FUNCTION_BLOCK FB_Slitter EXTENDS FB_BASE IMPLEMENTS I_UnitState
VAR_INPUT
	Batch		: ULINT;
	Inspect		: BOOL;					// run routine without cut; just inspect
	InspectCmd	: ST_InspectCommands;
	TubeHmi		: ST_TubeParameters;	// used for manual commands
END_VAR
VAR_IN_OUT
	Tube		: ST_TubeParameters;
END_VAR
VAR_OUTPUT 
	FilesLoaded		: BOOL;
	BatchOut		: ULINT;
	CounterOut		: ULINT;
	CountFailedOut	: UINT;
	Status			: INT; 	// 0 = idle, 1 = processing, 2 = pass, 3 = fail, 4 = no detect
END_VAR
VAR
	Mandrel				: FB_Mandrel;
	MandrelParameters	: ST_MandrelParameters;
	Camera				: FB_Camera;
	CameraParameters	: ST_CameraParameters;
	Cutter				: FB_Cutter;
	CutterParameters 	: ST_CutterParameters;
	Ejector				: FB_Ejector;
	EjectorParameters	: ST_EjectorParameters;
	EjectState			: INT;
	Eject				: BOOL;
	
	Manual		: ST_ManualCommands;
	bBusy		: BOOL;	
	bCalibration: BOOL;
	strJobName	: STRING;	// for manual override of which camera program is used
	nIndex		: INT;
	PreviousTubeIndex	: INT;
	fbFileOpen	: FB_FileOpen;
	fbFileWrite	: FB_FileWrite;
	fbFileClose	: FB_FileClose;
	fbLocalSystemTime	: FB_LocalSystemTime;
	bDecrementSpindle: BOOL;
	bIncrementSpindle: BOOL;
	bInspect: BOOL;
	bInspectComplete: BOOL;
	nCalibrationCounter : INT;
	CalibrationArrayX	: ARRAY[0..CalMax] OF LREAL;
	CalibrationArrayY	: ARRAY[0..CalMax] OF LREAL;
	AverageX 			: LREAL;
	AverageY 			: LREAL;
	
	fbXmlSrvRead		: FB_XmlSrvRead;
	fbXmlSrvWrite		: FB_XmlSrvWrite;

	fbMessageSaved		: FB_TcMessage;
		
END_VAR
VAR CONSTANT
	CalMax	: INT := 9;
END_VAR
VAR PERSISTENT
	Counter		: UINT;
	CountFailed	: UINT;
END_VAR


SUPER^();

IF eState <> E_PMLState.ePMLState_Undefined THEN
	Mandrel.MonitorParameters();
	Camera.MonitorParameters();
	Cutter.MonitorParameters();
	Ejector.MonitorParameters();
END_IF

Mandrel.ConvertVaccum();
Mandrel.TubeParameters := Tube;

IF Batch <> BatchOut THEN
	BatchOut := Batch;
	Counter := 0;
	CountFailed := 0;
END_IF

CounterOut := Counter;
CountFailedOut := CountFailed;

Camera.TubeParameters := Tube;

CASE eState OF
	E_PMLState.ePMLState_Idle: Status := 0;
	E_PMLState.ePMLState_Starting: Status := 1;
	(* put in executing to get fast answer - don't wait for execute to finish
	E_PMLState.ePMLState_Completing:
		IF Camera.Pass THEN
			Status := 2;
		ELSIF Camera.Fail THEN
			Status := 3;
		ELSIF ...
			Status := 4;
		END_IF
	*)
END_CASE

METHOD FB_init : BOOL
VAR_INPUT
	bInitRetains : BOOL; // if TRUE, the retain variables are initialized (warm start / cold start)
	bInCopyCode : BOOL;  // if TRUE, the instance afterwards gets moved into the copy code (online change)
END_VAR
IF NOT fbMessageSaved.EqualsToEventEntryEx(stOther := TC_EVENTS.SlitterEvents.ParametersSaved) THEN
	fbMessageSaved.CreateEx(TC_EVENTS.SlitterEvents.ParametersSaved, 0);
END_IF
END_METHOD

METHOD M_Aborting
M_StateComplete();

bBusy := FALSE;
bCalibration := FALSE;
Cutter.Abort();
Ejector.Abort();
Mandrel.Abort();
M_CalibrateCamera(Execute := FALSE);
Eject := FALSE;
EjectState := 0;
nCalibrationCounter := 0;

Manual.bCameraCalibrate := FALSE;
Manual.bCameraComputePeak := FALSE;
Manual.bCameraInspect := FALSE;
Manual.bCameraRawData := FALSE;
Manual.bCameraTrigger := FALSE;
Manual.bCutSample := FALSE;
Manual.bCutterDisable := FALSE;
Manual.bCutterHome := FALSE;
Manual.bCutterMoveAbs := FALSE;
Manual.bCutterReset := FALSE;
Manual.bEjectAxisEnableToggle := FALSE;
Manual.bEjectAxisFailPosition := FALSE;
Manual.bEjectAxisHomePosition := FALSE;
Manual.bEjectAxisPassPosition := FALSE;
Manual.bEjectAxisReset := FALSE;
Manual.bEjectBlowOff := FALSE;
Manual.bEjectReset := FALSE;
Manual.bEjectSamplePass := FALSE;
Manual.bEjectSampleFail := FALSE;
Manual.bEjectVacuum := FALSE;
Manual.bEjectZExtend := FALSE;
Manual.bEjectZNeutral := FALSE;
Manual.bEjectZOff := FALSE;
Manual.bEjectZRetract := FALSE;
Manual.bLowerMandrel := FALSE;
Manual.bMandrelReset := FALSE;
Manual.bMandrelSpindleRotate := FALSE;
Manual.bMandrelSpindleToggle := FALSE;
Manual.bMandrelXEnableToggle := FALSE;
Manual.bMandrelYEnableToggle := FALSE;
Manual.bMoveToCutPosition := FALSE;
Manual.bMoveToEjectPosition := FALSE;
Manual.bMoveToInspectPosition := FALSE;
Manual.bMoveToLoadPosition := FALSE;
Manual.bRaiseMandrel := FALSE;
Manual.bSaveMandrelParameters := FALSE;
Manual.bToggleMandrelVacuum := FALSE;
Manual.bVacuumAxisToggleEnable := FALSE;
Manual.bVacuumAxisMove := FALSE;
Manual.bVacuumAxisReset := FALSE;
END_METHOD

METHOD M_CalibrateCamera : INT;
VAR_INPUT
	Execute			: BOOL;
END_VAR
VAR_INST
	rTrig			: R_TRIG;
	nIndex			: INT;
	Position		: LREAL;
	debug			: INT;
	debug1			: INT;
	debug2			: INT;
END_VAR
rTrig(CLK := Execute);
IF rTrig.Q THEN
	nIndex := 10;
	Mandrel.MoveToInspectPosition(Execute := FALSE, InspectPositionX := Tube.InspectPositionX, InspectPositionY := Tube.InspectPositionY);
	Mandrel.MoveToLoadPosition(Execute := FALSE);
	Mandrel.MoveXAbs(Execute := FALSE, Position := 0);
	Mandrel.MoveYAbs(Execute := FALSE, Position := 0);
	Camera.TriggerCamera(Execute := FALSE);
	bCalibration := TRUE;
END_IF

IF NOT Execute THEN
	debug := debug + 1;
	nIndex := 0;
END_IF

CASE nIndex OF
	0: // idle state
		M_CalibrateCamera := 0;
		bCalibration := FALSE;
	10: // move to first inspection position
		IF Mandrel.MoveToInspectPosition(Execute := TRUE, InspectPositionX := Tube.InspectPositionX, InspectPositionY := Tube.InspectPositionY) = 1 THEN
			Mandrel.MoveToInspectPosition(Execute := FALSE, InspectPositionX := Tube.InspectPositionX, InspectPositionY := Tube.InspectPositionY);
			nIndex := 20;
		ELSIF Mandrel.MoveToInspectPosition(Execute := TRUE, InspectPositionX := Tube.InspectPositionX, InspectPositionY := Tube.InspectPositionY) = -1 THEN
			Mandrel.MoveToInspectPosition(Execute := FALSE, InspectPositionX := Tube.InspectPositionX, InspectPositionY := Tube.InspectPositionY);
			nIndex := 100;
		END_IF
	20: // trigger the camera
		IF Camera.TriggerCamera(Execute := TRUE) THEN
			Camera.PatternX1 := Camera.PatternMatchX;
			Camera.PatternY1 := Camera.PatternMatchY;
			Camera.TriggerCamera(Execute := FALSE);
			nIndex := 30;
		END_IF
	30: // move to second position in x
		Position := Tube.InspectPositionX + Camera.CalibrationDistance; 
		IF Mandrel.MoveXAbs(Execute := TRUE, Position := Position) = 1 THEN
			Mandrel.MoveXAbs(Execute := FALSE, Position := Position);
			nIndex := 40;
		ELSIF Mandrel.MoveXAbs(Execute := TRUE, Position := Position) = -1 THEN
			Mandrel.MoveXAbs(Execute := FALSE, Position := Position);
			nIndex := 100;
		END_IF
	40: // trigger the camera
		IF Camera.TriggerCamera(Execute := TRUE) THEN
			Camera.PatternX2 := Camera.PatternMatchX;
			Camera.PatternY2 := Camera.PatternMatchY;
			Camera.TriggerCamera(Execute := FALSE);
			nIndex := 50;
		END_IF
	45: // 
		Mandrel.MoveYAbs(Execute := FALSE, Position := 0);
		nIndex := 50;
	50: // move to the third position in y
		Position := Tube.InspectPositionY + Camera.CalibrationDistance; 
		IF Mandrel.MoveYAbs(Execute := TRUE, Position := Position) = 1 THEN
			Mandrel.MoveYAbs(Execute := FALSE, Position := Position);
			nIndex := 60;
		ELSIF Mandrel.MoveYAbs(Execute := TRUE, Position := Position) = -1 THEN
			Mandrel.MoveYAbs(Execute := FALSE, Position := Position);
			nIndex := 100;
		END_IF
	60: // trigger camera
		IF Camera.TriggerCamera(Execute := TRUE) THEN
			Camera.PatternX3 := Camera.PatternMatchX;
			Camera.PatternY3 := Camera.PatternMatchY;
			Camera.TriggerCamera(Execute := FALSE);
			nIndex := 70;
		END_IF
	70: // Calculate the pitch
		Camera.Calibrate();
		nIndex := 80; 
	80: // return to load position	
		IF Mandrel.MoveToLoadPosition(Execute := TRUE) <> 0 THEN
			Mandrel.MoveToLoadPosition(Execute := FALSE);
			nIndex := 90;
		END_IF
	90: // done state
		M_CalibrateCamera := 1;
	 
	100: // error state
		M_CalibrateCamera := -1;
	
END_CASE
END_METHOD

METHOD M_Clearing
CASE eMode OF
	E_PMLProtectedUnitMode.ePMLProtUnitMode_Manual: M_ClearingManual();
	
	E_PMLProtectedUnitMode.ePMLProtUnitMode_Production: M_ClearingProduction();
END_CASE
END_METHOD

METHOD M_ClearingManual : BOOL
VAR_INPUT
END_VAR
M_StateComplete();
//M_ClearingManual := TRUE;
END_METHOD

METHOD M_ClearingProduction : BOOL
VAR_INPUT
END_VAR
CASE nState OF
	0:	// reset the variables
		Mandrel.Clear(Execute := FALSE);
		Cutter.Clear(Execute := FALSE);
		Ejector.Reset(Execute := FALSE);
		nState := 10;
	10: // reset the cutter
		IF Cutter.Clear(Execute := TRUE) = 1 THEN
			Cutter.Clear(Execute := FALSE);
			nState := 20;
		END_IF	
	20: // reset the ejector
		IF Ejector.Reset(Execute := TRUE) = 1 THEN
			Ejector.Reset(Execute := FALSE);
			nState := 30;		END_IF

	30: // reset the different objects
		IF Mandrel.Clear(Execute := TRUE) = 1 THEN
			Mandrel.Clear(Execute := FALSE);
			nState := 40;
		END_IF
	40:	// done state
		M_StateComplete();
END_CASE
END_METHOD


METHOD M_Complete
END_METHOD

METHOD M_Completing

VAR
	EjectSample: INT;
END_VAR
IF eMode = E_PMLProtectedUnitMode.ePMLProtUnitMode_Production THEN
	CASE EjectState OF
		0: // wait for eject command
			M_StateComplete();
		10: // execute the eject pass sequence
			EjectSample := Ejector.EjectSamplePass(Execute := TRUE);
			IF EjectSample = 1 THEN
				Eject := FALSE;
				Ejector.EjectSamplePass(Execute := FALSE);
				EjectState := 0;
			ELSIF EjectSample = -1 THEN
				Eject := FALSE;
				EjectState := 0;
				Ejector.EjectSamplePass(Execute := FALSE);
			END_IF
		20: // execute the eject fail sequence
			EjectSample := Ejector.EjectSampleFail(Execute := TRUE);
			IF EjectSample = 1 THEN
				Eject := FALSE;
				Ejector.EjectSampleFail(Execute := FALSE);
				EjectState := 0;
			ELSIF EjectSample = -1 THEN
				Eject := FALSE;
				EjectState := 0;
				Ejector.EjectSampleFail(Execute := FALSE);
			END_IF
	END_CASE
ELSE
	M_StateComplete();
END_IF
END_METHOD

METHOD M_Execute
VAR_INST
	Result					: INT;
END_VAR
VAR
	CutPositionY 			: LREAL;
	VelocityY 				: LREAL;
	MoveToCutPosition 		: INT;
	MoveToInspectPosition 	: INT;
	MoveToEjectPosition 	: INT;
	MoveToLoadPosition 		: INT;
	CutSample				: INT;
	EjectSample 			: INT;

	CameraIndex 			: INT;
	FileName				: STRING;
	FilePath				: STRING;
	RotateDistance			: LREAL;
END_VAR
VAR_INST
	StrResult				: STRING(255);
	SampleLowered			: BOOL;
	LiftTon					: TON := (PT := T#500MS);
	VacuumSensorTON			: TON := (PT := T#2S);
	hFile					: UINT;
	AttemptCounter			: INT;
	Pass					: BOOL;
	Message					: STRING(255);
END_VAR
Eject := FALSE;
fbLocalSystemTime(
	sNetId := '',
	bEnable := TRUE,
	dwCycle := 1);

IF eMode = E_PMLProtectedUnitMode.ePMLProtUnitMode_Production THEN
	CASE nState OF
		0: // do we need to write to the camera?
			AttemptCounter := 0;
			bDecrementSpindle:= FALSE;
			bIncrementSpindle:= FALSE;
			bInspect:= FALSE;
			bInspectComplete:= FALSE;

			SampleLowered := FALSE;
			VacuumSensorTON(IN := FALSE);
			Result := Camera.SelectCameraProgram(Execute := TRUE);
			IF Result = 1 THEN
				Camera.SelectCameraProgram(Execute := FALSE);
				nState := 5;
			ELSIF Result = -1 THEN
				Camera.SelectCameraProgram(Execute := FALSE);
				Message := 'Camera failed to read/write to modbus.';
				nState := 666;
			END_IF
		5: // move the vacuum axis to the correct location
			IF Mandrel.MoveToVacPosition(Execute := TRUE) THEN
				Mandrel.MoveToVacPosition(Execute := FALSE);
				nState := 10;
			END_IF
		10: // turn on mandrel vacuum and move to cut position
			Mandrel.MandrelVacuum := TRUE;
			IF Mandrel.LowerSample() = 1 THEN
				SampleLowered := TRUE;
				nState := 11;
			END_IF
		11: // wait for vacuum sensor to detect the tube
			VacuumSensorTON(IN := TRUE);
			IF Mandrel.VacuumSensor > Tube.VacuumThreshold THEN
				nState := 15;
				VacuumSensorTON(IN := FALSE);
			END_IF
			IF VacuumSensorTON.Q THEN
				Mandrel.MandrelVacuum := FALSE;
				nState := 110;
				VacuumSensorTON(IN := FALSE);
			END_IF
		15: // move to cut position
			MoveToCutPosition := Mandrel.MoveToCutPosition(Execute := TRUE, CutPositionX := Tube.CutPositionX, CutPositionY := Tube.CutPositionY);
			IF MoveToCutPosition = 1 AND SampleLowered THEN
				Mandrel.MoveToCutPosition(Execute := FALSE, CutPositionX := Tube.CutPositionX, CutPositionY := Tube.CutPositionY);
				nState := 20;
				SampleLowered := FALSE;
			ELSIF MoveToCutPosition = -1 THEN
				Mandrel.MoveToCutPosition(Execute := FALSE, CutPositionX := Tube.CutPositionX, CutPositionY := Tube.CutPositionY);
				nState := 666;
				Message := 'Mandrel failed to move.';
				SampleLowered := FALSE;
			END_IF
		20: // make a cut unless we are just inspecting
			IF Inspect THEN
				nState := 30;
			ELSE
				CutSample := Cutter.CutSample(Execute := TRUE);
				IF CutSample = 1 THEN
					Cutter.CutSample(Execute := FALSE);
					nState := 30;
				ELSIF CutSample = -1 THEN
					Cutter.CutSample(Execute := FALSE);
					nState := 666;
				END_IF
			END_IF
		30: // raise sample
			// move to inspect position
			Mandrel.LiftSample();
			MoveToInspectPosition := Mandrel.MoveToInspectPosition(Execute := TRUE, InspectPositionX := Tube.InspectPositionX, InspectPositionY := Tube.InspectPositionY);
			IF MoveToInspectPosition = 1 THEN
				Mandrel.MoveToInspectPosition(Execute := FALSE, InspectPositionX := Tube.InspectPositionX, InspectPositionY := Tube.InspectPositionY);
				nState := 35;
			ELSIF MoveToInspectPosition = -1 THEN
				Mandrel.MoveToInspectPosition(Execute := FALSE, InspectPositionX := Tube.InspectPositionX, InspectPositionY := Tube.InspectPositionY);
				nState := 666;
			END_IF
		35: // add 500 ms delay for lifter
			LiftTON.IN := TRUE;
			IF LiftTON.Q THEN
				LiftTON.IN := FALSE;
				IF Inspect THEN
					nState := 36;
				ELSE
					nState := 40;
				END_IF
			END_IF
			LiftTON();
		36: // Inspect under manual control
			Result := Camera.Inspect(Execute := TRUE);
			IF Result = 1 THEN
				nState := 37;
				Camera.Inspect(Execute := FALSE);
				IF Camera.Pass THEN
					Status := 2;
				ELSE
					Status := 3;
				END_IF
			ELSIF Result = -1 THEN
				Status := 4;
				nState := 37;
			END_IF
			//nState := 37;
		37: // wait for command
			IF bDecrementSpindle THEN
				bDecrementSpindle := FALSE;
				nState := 39;
			ELSIF bIncrementSpindle THEN
				bIncrementSpindle := FALSE;
				nState := 38;
			ELSIF bInspect THEN
				bInspect := FALSE;
				nState := 36;
			ELSIF bInspectComplete THEN
				bInspectComplete := FALSE;
				nState := 70;
			END_IF
		38: // increment spindle
			IF Mandrel.RotateSpindle(Execute := TRUE, Distance := Mandrel.SpindleIncrement ) <> 0 THEN
				Mandrel.RotateSpindle(Execute := FALSE, Distance := Mandrel.SpindleIncrement);
				nState := 37;
			END_IF
		39: // decrement spindle
			IF Mandrel.RotateSpindle(Execute := TRUE, Distance := -1 * Mandrel.SpindleIncrement) <> 0 THEN
				Mandrel.RotateSpindle(Execute := FALSE, Distance := -1 * Mandrel.SpindleIncrement);
				nState := 37;
			END_IF
			
		40: // inspect
			Result := Camera.Inspect(Execute := TRUE);
			IF Result = 1 THEN
				Camera.Inspect(Execute := FALSE);
				IF Camera.Pass THEN
					Mandrel.MandrelVacuum := FALSE;
					IF Manual.bCalibrateMandrel THEN
						CalibrationArrayX[nCalibrationCounter] := Camera.DeltaXmmWithOffset;
						CalibrationArrayY[nCalibrationCounter] := Camera.DeltaYmmWithOffset;
						nCalibrationCounter := nCalibrationCounter + 1;
						IF nCalibrationCounter > CalMax THEN
							MandrelCalibration();
							Manual.bCalibrateMandrel := FALSE;
							nCalibrationCounter := 0;
						END_IF
					END_IF
					Pass := TRUE;
					nState := 50;	// passed -> go to eject pass station
					Status := 2;
				ELSE
					Mandrel.MandrelVacuum := FALSE;
					Pass := FALSE;
					nState := 50;	// failed -> go to eject fail station
					Status := 3;
				END_IF
			ELSIF Result = -1 THEN	// couldn't find the pattern; need to advance the counter and retry
				AttemptCounter := AttemptCounter + 1;
				Camera.Inspect(Execute := FALSE);
				IF AttemptCounter > 3 THEN	// error
					nState := 70;			// error out
					Status := 4;
				ELSE						// advance the motor a bit and retry
					nState := 45;
				END_IF
			END_IF
		45: // advance the tube a bit and then go and retry the process
			Result := Mandrel.MoveXRel(Execute := TRUE, Distance := 1);
			IF Result = 1 THEN
				Mandrel.MoveXRel(Execute := FALSE, Distance := 1);
				nState := 35;
			END_IF
			
		50: // move to eject position		
			MoveToEjectPosition := Mandrel.MoveToEjectPosition(Execute := TRUE, EjectPositionX := Tube.EjectPositionX, EjectPositionY := Tube.EjectPositionY);
			IF MoveToEjectPosition = 1 THEN
				Mandrel.MoveToEjectPosition(Execute := FALSE, EjectPositionX := Tube.EjectPositionX, EjectPositionY := Tube.EjectPositionY);
				nState := 60;
			ELSIF MoveToEjectPosition = -1 THEN
				Mandrel.MoveToEjectPosition(Execute := FALSE, EjectPositionX := Tube.EjectPositionX, EjectPositionY := Tube.EjectPositionY);
				nState := 666;
			END_IF
		60: // do the eject sequence 
			Eject := TRUE;		
			// wait for the system to retract
			IF Ejector.IsEjectZExtend THEN
				nState := 65;
			END_IF
		65: // wait for ejector actuator to be clear to retract the mandrel
			IF Ejector.IsEjectZRetract THEN
				nState := 70;
			END_IF 
		70: // move to load position
			Mandrel.MandrelVacuum := FALSE;

			IF Mandrel.LowerSample() = 1 THEN
				SampleLowered := TRUE;
			END_IF
			IF Manual.bCalibrateMandrel THEN
				IF Mandrel.SpindleOffset >= 0 THEN
					RotateDistance := (360.0 / (INT_TO_LREAL(CalMax)+1.0)) - Mandrel.SpindleOffset;
				ELSE
					RotateDistance := -1 * ( (360.0 / (INT_TO_LREAL(CalMax)+1.0)) + Mandrel.SpindleOffset);
				END_IF
				IF Mandrel.RotateSpindle(Execute := TRUE, Distance := RotateDistance) <> 0 THEN
					Mandrel.RotateSpindle(Execute := FALSE, Distance := RotateDistance);
					nState := 75;
				END_IF
			ELSE
				nState := 75;			
			END_IF
		75: // move to load position cont'd
			IF Mandrel.LowerSample() = 1 THEN
				SampleLowered := TRUE;
			END_IF

			MoveToLoadPosition := Mandrel.MoveToLoadPosition(Execute := TRUE);
			IF MoveToLoadPosition = 1 AND SampleLowered THEN
				Mandrel.MoveToLoadPosition(Execute := FALSE);
				SampleLowered := FALSE;
				nState := 80;
			ELSIF MoveToLoadPosition = -1 THEN
				SampleLowered := FALSE;
				Mandrel.MoveToLoadPosition(Execute := FALSE);
				nState := 666;
			END_IF
		80: // check if vacuum is off
			IF Mandrel.VacuumSensor < Tube.VacuumThreshold THEN
				nState := 90;
				Mandrel.MandrelVacuum := FALSE;
			END_IF
		90:	// increment counters state
			IF NOT Inspect THEN			
				Counter := Counter + 1;
				IF NOT Camera.Pass THEN
					CountFailed := CountFailed + 1;
				END_IF
				nState := 100;
			ELSE
				nState := 110;
			END_IF			
		100: // save to file
			FileName := CONCAT(ULINT_TO_STRING(Batch), '.txt');
			FilePath := CONCAT('D:\',FileName);
			fbFileOpen(
				sNetId := '',
				sPathName := FilePath,
				nMode := FOPEN_MODEAPPEND,
				ePath := E_OpenPath.PATH_GENERIC,
				hFile => hFile,
				bExecute := TRUE);
			IF NOT fbFileOpen.bBusy THEN
				fbFileOpen(
					sNetId := '',
					sPathName := FilePath,
					nMode := FOPEN_MODEAPPEND,
					ePath := E_OpenPath.PATH_GENERIC,
					bExecute := FALSE);
				nState := 101;
			END_IF
			IF fbFileOpen.bError THEN
				fbFileOpen(
					sNetId := '',
					sPathName := FilePath,
					nMode := FOPEN_MODEAPPEND,
					ePath := E_OpenPath.PATH_GENERIC,
					bExecute := FALSE);
				nState := 102;				
			END_IF
		101: // write data to file	
			StrResult := '';		
			StrResult := CONCAT(ULINT_TO_STRING(Batch), ', ');
			StrResult := CONCAT(StrResult, UINT_TO_STRING(Counter));
			StrResult := CONCAT(StrResult, ', ');
			// add the system time
			IF fbLocalSystemTime.bValid THEN
				StrResult := CONCAT(StrResult, SYSTEMTIME_TO_STRING(fbLocalSystemTime.systemTime));
				StrResult := CONCAT(StrResult, ', ');
			END_IF
			IF Camera.Pass THEN
				StrResult := CONCAT(StrResult, 'PASS, ');
			ELSIF Camera.Fail THEN
				StrResult := CONCAT(StrResult, 'FAIL, ');
			ELSIF Camera.NoDetect THEN
				StrResult := CONCAT(StrResult, 'NO DETECT, ');
			END_IF
			IF NOT Camera.NoDetect THEN
				StrResult := CONCAT(StrResult, 'x := ');
				StrResult := CONCAT(StrResult, REAL_TO_STRING(Camera.DeltaXmmWithOffset));
				StrResult := CONCAT(StrResult, ', y := ');
				StrResult := CONCAT(StrResult, REAL_TO_STRING(Camera.DeltaYmmWithOffset));
				StrResult := CONCAT(StrResult, ', length := ');
				StrResult := CONCAT(StrResult, REAL_TO_STRING(Camera.CutLengthWithOffset));
			ELSE
				StrResult := CONCAT(StrResult, 'x := not detected');
				StrResult := CONCAT(StrResult, ', y := not detected');
				StrResult := CONCAT(StrResult, ', length := not detected');			
			END_IF
			StrResult := CONCAT(StrResult, '$r$n');
			fbFileWrite(
				sNetId := '',
				hFile := hFile,
				pWriteBuff := ADR(StrResult),
				cbWriteLen := INT_TO_UINT(LEN(StrResult)),
				bExecute := TRUE
			);
			IF NOT fbFileWrite.bBusy THEN
				nState := 102;
				fbFileWrite(bExecute := FALSE);
			END_IF
			IF fbFileWrite.bError THEN
				nState := 102;
				fbFileWrite(bExecute := FALSE);
			END_IF
		102: // file close
			fbFileClose(
				sNetId := '',
				hFile := hFile,
				bExecute := TRUE);
			IF NOT fbFileClose.bBusy THEN
				fbFileClose(bExecute := FALSE);
				nState := 110;
			END_IF
			IF fbFileClose.bError THEN
				fbFileClose(bExecute := FALSE);
				nState := 110;
			END_IF
		110: // done state
			M_StateComplete();
	END_CASE
	
	CASE EjectState OF
		0: // wait for eject command
			Ejector.EjectSamplePass(Execute := FALSE);
			Ejector.EjectSampleFail(Execute := FALSE);
			IF Eject AND Pass THEN
				EjectState := 10;
			ELSIF Eject AND NOT Pass THEN
				EjectState := 20;
			END_IF
		10: // execute the eject pass sequence
			EjectSample := Ejector.EjectSamplePass(Execute := TRUE);
			IF EjectSample = 1 THEN
				Eject := FALSE;
				Ejector.EjectSamplePass(Execute := FALSE);
				EjectState := 0;
			ELSIF EjectSample = -1 THEN
				Eject := FALSE;
				EjectState := 0;
				Ejector.EjectSamplePass(Execute := FALSE);
			END_IF
		20: // execute the eject fail sequence
			EjectSample := Ejector.EjectSampleFail(Execute := TRUE);
			IF EjectSample = 1 THEN
				Eject := FALSE;
				Ejector.EjectSampleFail(Execute := FALSE);
				EjectState := 0;
			ELSIF EjectSample = -1 THEN
				Eject := FALSE;
				EjectState := 0;
				Ejector.EjectSampleFail(Execute := FALSE);
			END_IF

	END_CASE
ELSIF eMode = E_PMLProtectedUnitMode.ePMLProtUnitMode_Manual THEN
	M_Manual();
END_IF
END_METHOD


METHOD M_Held
END_METHOD


METHOD M_Holding
END_METHOD


METHOD M_Idle
END_METHOD

METHOD M_Manual : BOOL
VAR_INPUT
END_VAR
VAR_INST
	Operational	: BOOL;
	Result		: INT;
	TON			: TON := (PT := T#5S);
	x			: INT;
END_VAR

IF Manual.bCameraCalibrate THEN
	bBusy := TRUE;
	IF M_CalibrateCamera(Execute := TRUE) <> 0 THEN
		M_CalibrateCamera(Execute := FALSE);
		bBusy := FALSE;
		Manual.bCameraCalibrate := FALSE;
	END_IF
END_IF

IF Manual.bCameraComputePeak THEN
	bBusy := TRUE;
	IF Camera.Compute(Execute := TRUE) = 1 THEN
		bBusy := FALSE;
		Camera.Compute(Execute := FALSE);
		Manual.bCameraComputePeak := FALSE;
	END_IF
END_IF

IF Manual.bCameraInspect THEN
	bBusy := TRUE;
	IF Camera.Inspect(Execute := TRUE) = 1 THEN
		Camera.Inspect(Execute := FALSE);
		Manual.bCameraInspect := FALSE;
		bBusy := FALSE;
	END_IF
END_IF	

IF Manual.bCameraRawData THEN
	bBusy := TRUE;
	IF Camera.GetCameraData() <> 0 THEN
		bBusy := FALSE;
		Manual.bCameraRawData := FALSE;
	END_IF
END_IF

IF Manual.bCameraSelectTube THEN
	bBusy := TRUE;
	Result := Camera.SelectCameraProgram(Execute := TRUE);
	IF Result = 1 THEN
		bBusy := FALSE;
		Manual.bCameraSelectTube := FALSE;
		Camera.SelectCameraProgram(Execute := FALSE);
	ELSIF Result = -1 THEN
		bBusy := FALSE;
		Manual.bCameraSelectTube := FALSE;
		Camera.SelectCameraProgram(Execute := FALSE);
		x := x + 1;
	END_IF
END_IF

IF Manual.bCameraTrigger THEN
	bBusy := TRUE;
	IF Camera.TriggerCamera(Execute := TRUE) THEN
		Camera.TriggerCamera(Execute := FALSE);
		bBusy := FALSE;
		Manual.bCameraTrigger := FALSE;
	END_IF
END_IF

IF Manual.bCutSample THEN
	bBusy := TRUE;
	IF Cutter.CutSample(Execute := TRUE) <> 0 THEN
		Cutter.CutSample(Execute := FALSE);
		Manual.bCutSample := FALSE;
		bBusy := FALSE;
	END_IF
END_IF

IF Manual.bCutterDisable THEN
	IF NOT bBusy THEN
		Operational := Cutter.IsEnabled;
		TON(IN := TRUE);
	END_IF
	bBusy := TRUE;
	IF Operational THEN
		IF Cutter.Disable() THEN
			TON(IN := FALSE);
			bBusy := FALSE;
			Manual.bCutterDisable := FALSE;
		END_IF
	ELSE
		IF Cutter.Enable() OR TON.q	THEN
			bBusy := FALSE;
			TON(IN := FALSE);
			Manual.bCutterDisable := FALSE;
		END_IF
	END_IF
	TON();
END_IF

IF Manual.bCutterHome THEN
	bBusy := TRUE;
	IF Cutter.Home(Execute := TRUE) <> 0 THEN
		bBusy := FALSE;
		Cutter.Home(Execute := FALSE);
		Manual.bCutterHome := FALSE;
	END_IF
END_IF

IF Manual.bCutterMoveAbs THEN
	bBusy := FALSE;
	IF Cutter.MoveAbs(Execute := TRUE) <> 0 THEN
		bBusy := FALSE;
		Cutter.MoveAbs(Execute := FALSE);
		Manual.bCutterMoveAbs := FALSE;
	END_IF
END_IF

IF Manual.bCutterReset THEN
	bBusy := TRUE;
	IF Cutter.Reset(Execute := TRUE) <> 0 THEN
		bBusy := FALSE;
		Manual.bCutterReset := FALSE;
		Cutter.Reset(Execute := FALSE);
	END_IF
END_IF

IF Manual.bEjectBlowOff THEN
	Ejector.BlowOff := NOT Ejector.BlowOff;
	Manual.bEjectBlowOff := FALSE;
END_IF

IF Manual.bEjectSamplePass THEN
	bBusy := TRUE;
	IF Ejector.EjectSamplePass(Execute := TRUE) = 1 THEN
		Ejector.EjectSamplePass(Execute := FALSE);
		Manual.bEjectSamplePass := FALSE;
		bBusy := FALSE;
	END_IF
END_IF

IF Manual.bEjectSampleFail THEN
	bBusy := TRUE;
	IF Ejector.EjectSampleFail(Execute := TRUE) = 1 THEN
		Ejector.EjectSampleFail(Execute := FALSE);
		Manual.bEjectSampleFail := FALSE;
		bBusy := FALSE;
	END_IF
END_IF

IF Manual.bEjectVacuum THEN
	Ejector.PickUpVacuum := NOT Ejector.PickUpVacuum;
	Manual.bEjectVacuum := FALSE;
END_IF
(*
	bEjectAxisPassPosition	: BOOL;
	bEjectAxisHomePosition	: BOOL;
	bEjectAxisFailPosition	: BOOL;
	bEjectAxisEnable		: BOOL;
	bEjectAxisDisabe		: BOOL;
	bEjectAxisReset			: BOOL;
	bEjectSamplePass		: BOOL;
	bEjectSampleFail		: BOOL;
*)
IF Manual.bEjectAxisEnableToggle THEN
	IF NOT bBusy THEN
		Operational := Ejector.axis.IsEnabled;
	END_IF
	bBusy := TRUE;
	IF Operational THEN
		IF Ejector.axis.Disable() THEN
			bBusy := FALSE;
			Manual.bEjectAxisEnableToggle := FALSE;
		END_IF
	ELSE
		IF Ejector.axis.Enable() THEN
			bBusy := FALSE;
			Manual.bEjectAxisEnableToggle := FALSE;
		END_IF		
	END_IF
END_IF

IF Manual.bEjectAxisFailPosition THEN
	bBusy := TRUE;
	IF Ejector.axis.AbsMove(Execute := TRUE, 
		Position := Ejector.EjectAxisFailPosition, 
		Velocity := Ejector.EjectAxisVelocity) THEN
			Ejector.axis.AbsMove(Execute := FALSE, Position := Ejector.EjectAxisFailPosition, Velocity := Ejector.EjectAxisVelocity);	
			bBusy := FALSE;
			Manual.bEjectAxisFailPosition := FALSE;
	END_IF
END_IF

IF Manual.bEjectAxisHomePosition THEN
	bBusy := TRUE;
	IF Ejector.axis.AbsMove(Execute := TRUE, 
		Position := Ejector.EjectAxisHomePosition, 
		Velocity := Ejector.EjectAxisVelocity) THEN
			Ejector.axis.AbsMove(Execute := FALSE, Position := Ejector.EjectAxisHomePosition, Velocity := Ejector.EjectAxisVelocity);
			bBusy := FALSE;
			Manual.bEjectAxisHomePosition := FALSE;
	END_IF
END_IF

IF Manual.bEjectAxisPassPosition THEN
	bBusy := TRUE;
	IF Ejector.axis.AbsMove(Execute := TRUE, 
		Position := Ejector.EjectAxisPassPosition, 
		Velocity := Ejector.EjectAxisVelocity) THEN
			Ejector.axis.AbsMove(Execute := FALSE, Position := Ejector.EjectAxisPassPosition, Velocity := Ejector.EjectAxisVelocity);
			bBusy := FALSE;
			Manual.bEjectAxisPassPosition := FALSE;
	END_IF
END_IF

IF Manual.bEjectAxisReset THEN
	bBusy := TRUE;
	IF Ejector.axis.Reset(Execute := TRUE) THEN
		Ejector.axis.Reset(Execute := FALSE);
		bBusy := FALSE;
		Manual.bEjectAxisReset := FALSE;
	END_IF
END_IF

IF Manual.bEjectReset THEN
	bBusy := TRUE;
	IF Ejector.Reset(TRUE) = 1 THEN
		Ejector.Reset(FALSE);
		bBusy := FALSE;
		Manual.bEjectReset := FALSE;
	END_IF
END_IF

IF Manual.bEjectZExtend THEN
	bBusy := TRUE;
	IF Ejector.zSlide.Extend() = 1 THEN
		bBusy := FALSE;
		Manual.bEjectZExtend := FALSE;
	END_IF
END_IF

IF Manual.bEjectZNeutral THEN
	bBusy := TRUE;
	IF Ejector.zSlide.Neutral() THEN
		bBusy := FALSE;
		Manual.bEjectZNeutral := FALSE;
	END_IF
END_IF

IF Manual.bEjectZRetract THEN
	bBusy := TRUE;
	IF Ejector.zSlide.Retract() = 1 THEN
		bBusy := FALSE;
		Manual.bEjectZRetract := FALSE;
	END_IF
END_IF

IF Manual.bLowerMandrel THEN
	bBusy := TRUE;
	IF Mandrel.LowerSample() = 1 THEN
		bBusy := FALSE;
		Manual.bLowerMandrel := FALSE;
	END_IF
END_IF

IF Manual.bMandrelSpindleRotate THEN
	bBusy := TRUE;
	IF Mandrel.RotateSpindle(Execute := TRUE, Distance := Mandrel.SpindleIncrement) <> 0 THEN
		bBusy := FALSE;
		Mandrel.RotateSpindle(Execute := FALSE, Distance := Mandrel.SpindleIncrement);
		Manual.bMandrelSpindleRotate := FALSE;
	END_IF
END_IF

IF Manual.bMandrelSpindleToggle THEN
	IF NOT bBusy THEN
		Operational := Mandrel.OperationalSpindle;
	END_IF
	bBusy := TRUE;
	IF Operational THEN
		IF Mandrel.DisableSpindle() THEN
			bBusy := FALSE;
			Manual.bMandrelSpindleToggle := FALSE;
		END_IF
	ELSE
		IF Mandrel.EnableSpindle() THEN
			bBusy := FALSE;
			Manual.bMandrelSpindleToggle := FALSE;
		END_IF
	END_IF
END_IF

IF Manual.bMandrelXEnableToggle THEN
	IF NOT bBusy THEN
		Operational := Mandrel.OperationalX;
	END_IF
	bBusy := TRUE;
	IF Operational THEN
		IF Mandrel.DisableX() THEN
			bBusy := FALSE;
			Manual.bMandrelXEnableToggle := FALSE;
		END_IF
	ELSE
		IF Mandrel.EnableX() THEN
			bBusy := FALSE;
			Manual.bMandrelXEnableToggle := FALSE;
		END_IF
	END_IF	
END_IF

IF Manual.bMandrelYEnableToggle THEN
	IF NOT bBusy THEN
		Operational := Mandrel.OperationalY;
	END_IF
	bBusy := TRUE;
	IF Operational THEN
		IF Mandrel.DisableY() THEN
			bBusy := FALSE;
			Manual.bMandrelYEnableToggle := FALSE;
		END_IF
	ELSE
		IF Mandrel.EnableY() THEN
			bBusy := FALSE;
			Manual.bMandrelYEnableToggle := FALSE;
		END_IF
	END_IF		
END_IF

IF Manual.bMandrelReset THEN
	bBusy := TRUE;
	IF Mandrel.Reset(Execute := TRUE) = 1 THEN
		Mandrel.Reset(Execute := FALSE);
		bBusy := FALSE;
		Manual.bMandrelReset := FALSE;
	END_IF
END_IF

IF Manual.bMoveToCutPosition THEN
	bBusy := TRUE;
	IF Mandrel.MoveToCutPosition(Execute := TRUE, CutPositionX := TubeHmi.CutPositionX, CutPositionY := TubeHmi.CutPositionY ) = 1 THEN
		Mandrel.MoveToCutPosition(Execute := FALSE, CutPositionX := TubeHmi.CutPositionX, CutPositionY := TubeHmi.CutPositionY);
		Manual.bMoveToCutPosition := FALSE;
		bBusy := FALSE;
	END_IF
END_IF

IF Manual.bMoveToEjectPosition THEN
	bBusy := TRUE;
	IF Mandrel.MoveToEjectPosition(Execute := TRUE, EjectPositionX := TubeHmi.EjectPositionX, EjectPositionY := TubeHmi.EjectPositionY) = 1 THEN
		Mandrel.MoveToEjectPosition(Execute := FALSE, EjectPositionX := TubeHmi.EjectPositionX, EjectPositionY := TubeHmi.EjectPositionY);
		Manual.bMoveToEjectPosition := FALSE;
		bBusy := FALSE;
	END_IF
END_IF

IF Manual.bMoveToInspectPosition THEN
	bBusy := TRUE;
	IF Mandrel.MoveToInspectPosition(Execute := TRUE, InspectPositionX := TubeHmi.InspectPositionX, InspectPositionY := TubeHmi.InspectPositionY) = 1 THEN
		Mandrel.MoveToInspectPosition(Execute := FALSE, InspectPositionX := TubeHmi.InspectPositionX, InspectPositionY := TubeHmi.InspectPositionY);
		Manual.bMoveToInspectPosition := FALSE;
		bBusy := FALSE;
	END_IF
END_IF

IF Manual.bMoveToLoadPosition THEN
	bBusy := TRUE;
	IF Mandrel.MoveToLoadPosition(Execute := TRUE) = 1 THEN
		Mandrel.MoveToLoadPosition(Execute := FALSE);
		Manual.bMoveToLoadPosition := FALSE;
		bBusy := FALSE;
	END_IF
END_IF

IF Manual.bRaiseMandrel THEN
	bBusy := TRUE;
	IF Mandrel.LiftSample() = 1 THEN
		bBusy := FALSE;
		Manual.bRaiseMandrel := FALSE;
	END_IF
END_IF

IF Manual.bToggleMandrelVacuum THEN
	Mandrel.MandrelVacuum := NOT Mandrel.MandrelVacuum;
	Manual.bToggleMandrelVacuum := FALSE;
END_IF


IF Manual.bVacuumAxisMove THEN
	bBusy := TRUE;
	IF Mandrel.VacAxis.AbsMove(Execute := TRUE, Position := TubeHmi.VacPosition, Velocity := Mandrel.VacuumVelocity) THEN
		Mandrel.VacAxis.AbsMove(Execute := FALSE, Position := 0, Velocity := 0);
		bBusy := FALSE;
		Manual.bVacuumAxisMove := FALSE;
	END_IF
END_IF

IF Manual.bVacuumAxisReset THEN
	bBusy := TRUE;
	IF Mandrel.VacAxis.Reset(Execute := TRUE) THEN
		Mandrel.VacAxis.Reset(Execute := FALSE);
		bBusy := FALSE;
		Manual.bVacuumAxisReset := FALSE;
	END_IF
END_IF

IF Manual.bVacuumAxisToggleEnable THEN
	IF NOT bBusy THEN
		Operational := Mandrel.VacAxis.IsEnabled;
	END_IF
	bBusy := TRUE;
	IF Operational THEN
		IF Mandrel.VacAxis.Disable() THEN
			bBusy := FALSE;
			Manual.bVacuumAxisToggleEnable := FALSE;
		END_IF
	ELSE
		IF Mandrel.VacAxis.Enable() THEN
			bBusy := FALSE;
			Manual.bVacuumAxisToggleEnable := FALSE;
		END_IF
	END_IF
END_IF
END_METHOD

METHOD M_Production : BOOL
VAR_INPUT
END_VAR
END_METHOD

METHOD M_Resetting
M_StateComplete();
END_METHOD

METHOD M_Starting
Mandrel.MoveToCutPosition(Execute := FALSE, CutPositionX := Tube.CutPositionX, CutPositionY := Tube.CutPositionY);
Cutter.CutSample(Execute := FALSE);
Mandrel.MoveToInspectPosition(Execute := FALSE, InspectPositionX := Tube.InspectPositionX, InspectPositionY := Tube.InspectPositionY);
Camera.Inspect(Execute := FALSE);
Mandrel.MoveToEjectPosition(Execute := FALSE, EjectPositionX := Tube.EjectPositionX, EjectPositionY := Tube.EjectPositionY);
Mandrel.MoveToLoadPosition(Execute := FALSE);
Camera.SelectCameraProgram(Execute := FALSE);
//Mandrel.MoveToVacPosition(Execute := FALSE);
fbFileOpen(bExecute := FALSE);
fbFileWrite(bExecute := FALSE);
fbFileClose(bExecute := FALSE);

IF Mandrel.LowerSample() = 1 THEN
	M_StateComplete();
END_IF
END_METHOD


METHOD M_Stopped
END_METHOD


METHOD M_Stopping
END_METHOD


METHOD M_Suspended
END_METHOD


METHOD M_Suspending
END_METHOD


METHOD M_Undefined
END_METHOD


METHOD M_Unholding
END_METHOD


METHOD M_Unsuspending
END_METHOD

METHOD MandrelCalibration : BOOL
VAR_INPUT
END_VAR

VAR
	i: INT;
	SumX: LREAL;
	SumY: LREAL;
END_VAR
SumX := 0;
SumY := 0;
FOR i:= 0 TO CalMax DO
	SumX := CalibrationArrayX[i] + SumX;
	SumY := CalibrationArrayY[i] + SumY;
END_FOR
AverageX := SumX / 10.0;
AverageY := SumY / 10.0;

Tube.CutPositionX := Tube.CutPositionX - AverageX;
Tube.CutPositionY := Tube.CutPositionY - AverageY;
END_METHOD

PROPERTY MandrelVacuum : BOOL
GET
MandrelVacuum := Mandrel.MandrelVacuum;
END_GET
SET
Mandrel.MandrelVacuum := MandrelVacuum;
END_SET
END_PROPERTY

METHOD ReadParameters : BOOL
VAR_INPUT
	Execute	: BOOL;
END_VAR
VAR_INST
	nReadIndex	: INT;
	rTrig		: R_TRIG;
END_VAR
ReadParameters := FALSE;
rTrig(CLK := Execute);
IF rTrig.Q THEN
	nReadIndex := 5;
END_IF

IF NOT Execute THEN
	nReadIndex := 0;
END_IF

CASE nReadIndex OF
	5: // read the info from the config file for the camera
		fbXmlSrvRead.sXPath := '/Configuration/Camera';
		fbXmlSrvRead.pSymAddr := ADR(CameraParameters);
		fbXmlSrvRead.cbSymSize := SIZEOF(CameraParameters);
		fbXmlSrvRead.bExecute := TRUE;
		nReadIndex := 10;
	10: // wait for the info to load
		IF NOT fbXmlSrvRead.bBusy THEN
			fbXmlSrvRead.bExecute := FALSE;
			Camera.Parameters := CameraParameters;
			nReadIndex := 20;
		END_IF
	20: // read the info from the config file for the cutter
		fbXmlSrvRead.sXPath := '/Configuration/Cutter';
		fbXmlSrvRead.pSymAddr := ADR(CutterParameters);
		fbXmlSrvRead.cbSymSize := SIZEOF(CutterParameters);
		fbXmlSrvRead.bExecute := TRUE;
		nReadIndex := 30;
	30: // wait to complete
		IF NOT fbXmlSrvRead.bBusy THEN
			fbXmlSrvRead.bExecute := FALSE;
			Cutter.Parameters := CutterParameters;
			nReadIndex := 40;
		END_IF
	40: // read the ejector parameters
		fbXmlSrvRead.sXPath := '/Configuration/Ejector';
		fbXmlSrvRead.pSymAddr := ADR(EjectorParameters);
		fbXmlSrvRead.cbSymSize := SIZEOF(EjectorParameters);
		fbXmlSrvRead.bExecute := TRUE;
		nReadIndex := 50;
	50: // wait
		IF NOT fbXmlSrvRead.bBusy THEN
			fbXmlSrvRead.bExecute := FALSE;
			Ejector.Parameters := EjectorParameters;
			nReadIndex := 60;
		END_IF
	60: // read mandrel parameters
		fbXmlSrvRead.sXPath := '/Configuration/Mandrel';
		fbXmlSrvRead.pSymAddr := ADR(MandrelParameters);
		fbXmlSrvRead.cbSymSize := SIZEOF(MandrelParameters);
		fbXmlSrvRead.bExecute := TRUE;
		nReadIndex := 70;
	70: // wait
		IF NOT fbXmlSrvRead.bBusy THEN
			fbXmlSrvRead.bExecute := FALSE;
			Mandrel.Parameters := MandrelParameters;
			nReadIndex := 80;
		END_IF
	80: // done reading parameters
		ReadParameters := TRUE;		
END_CASE

fbXmlSrvRead(
	sNetId:= '', 
	ePath:= E_OpenPath.PATH_GENERIC, 
	nMode:= XMLSRV_SKIPMISSING, 
	sFilePath:= 'C:\Configuration.xml');
END_METHOD

METHOD SaveParameters : BOOL
VAR_INPUT
	Execute	: BOOL;
END_VAR
VAR_INST
	nSaveIndex	: INT;
	rTrig		: R_TRIG;
END_VAR
SaveParameters := FALSE;

rTrig(CLK := Execute);
IF rTrig.Q THEN
	nSaveIndex := 10;
END_IF

IF NOT Execute THEN
	nSaveIndex := 0;
END_IF

CASE nSaveIndex OF
	10: // read the info from the config file for the camera
		fbXmlSrvWrite.sXPath := '/Configuration/Camera';
		CameraParameters := Camera.Parameters;
		fbXmlSrvWrite.pSymAddr := ADR(CameraParameters);
		fbXmlSrvWrite.cbSymSize := SIZEOF(CameraParameters);
		fbXmlSrvWrite.bExecute := TRUE;
		nSaveIndex := 20;
	20: // wait for the info to load
		IF NOT fbXmlSrvWrite.bBusy THEN
			fbXmlSrvWrite.bExecute := FALSE;
			nSaveIndex := 30;
		END_IF
	30: // read the info from the config file for the cutter
		fbXmlSrvWrite.sXPath := '/Configuration/Cutter';
		CutterParameters := Cutter.Parameters;
		fbXmlSrvWrite.pSymAddr := ADR(CutterParameters);
		fbXmlSrvWrite.cbSymSize := SIZEOF(CutterParameters);
		fbXmlSrvWrite.bExecute := TRUE;
		nSaveIndex := 40;
	40: // wait to complete
		IF NOT fbXmlSrvWrite.bBusy THEN
			fbXmlSrvWrite.bExecute := FALSE;
			nSaveIndex := 50;
		END_IF
	50: // read the ejector parameters
		fbXmlSrvWrite.sXPath := '/Configuration/Ejector';
		EjectorParameters := Ejector.Parameters;
		fbXmlSrvWrite.pSymAddr := ADR(EjectorParameters);
		fbXmlSrvWrite.cbSymSize := SIZEOF(EjectorParameters);
		fbXmlSrvWrite.bExecute := TRUE;
		nSaveIndex := 60;
	60: // wait
		IF NOT fbXmlSrvWrite.bBusy THEN
			fbXmlSrvWrite.bExecute := FALSE;
			nSaveIndex := 70;
		END_IF
	70: // write mandrel parameters
		fbXmlSrvWrite.sXPath := '/Configuration/Mandrel';
		MandrelParameters := Mandrel.Parameters;
		fbXmlSrvWrite.pSymAddr := ADR(MandrelParameters);
		fbXmlSrvWrite.cbSymSize := SIZEOF(MandrelParameters);
		fbXmlSrvWrite.bExecute := TRUE;
		nSaveIndex := 80;
	80: // wait
		IF NOT fbXmlSrvWrite.bBusy THEN
			fbXmlSrvWrite.bExecute := FALSE;
			fbMessageSaved.Send(0);
			nSaveIndex := 90;
		END_IF
	90: // done writing parameters
		SaveParameters := TRUE;		
END_CASE

fbXmlSrvWrite(
	sNetId:= '', 
	ePath:= E_OpenPath.PATH_GENERIC, 
	nMode:= XMLSRV_SKIPMISSING, 
	sFilePath:= 'C:\Configuration.xml');
END_METHOD

END_FUNCTION_BLOCK

(* stored: Version 1.1.0.1, ProductVersion 3.1.4024.9
   POU FB_Slitter: Id {7a328348-b5d6-4092-afea-9c5e83fda193}, SpecialFunc None
   Method FB_init: Id {2695ce36-1c8e-4247-8301-5f66a071e9eb}
   Method M_Aborting: Id {90e7533a-87d1-4811-b79c-2aa2f3c4341d}
   Method M_CalibrateCamera: Id {50d870bc-07ae-4823-b6bc-a44278d18a58}
   Method M_Clearing: Id {7c5bba32-1fea-4eeb-a679-abf5c99e3b65}
   Method M_ClearingManual: Id {9afeb0de-b6ab-4a5c-b456-a2485d73aad8}
   Method M_ClearingProduction: Id {3443b4f9-432d-4c09-b717-0b592de4ed69}
   Method M_Complete: Id {1780f499-3e0b-4183-b06b-22e95e7c1e40}
   Method M_Completing: Id {a80dec61-c324-4326-8412-9c8115affa7f}
   Method M_Execute: Id {5a27d0f0-b578-4f5d-82aa-9f6a44f47776}
   Method M_Held: Id {f7964c5a-9ab2-4b03-b511-5669b80e790b}
   Method M_Holding: Id {2046f787-6bb5-45cd-8a99-c7ccdd803d21}
   Method M_Idle: Id {1739e9a5-6673-40a0-80d7-c3aaf63b68a4}
   Method M_Manual: Id {fcac7ef0-bbdb-4ad2-b9fa-ef6c3a9884c2}
   Method M_Production: Id {e87a4419-0c3b-4c97-a3dc-96de6ca8367a}
   Method M_Resetting: Id {daf711f7-219e-493a-bc7c-67b051c232c6}
   Method M_Starting: Id {35fd1ca4-1107-4a25-9fdf-221a14434d2d}
   Method M_Stopped: Id {41043cf7-9cd8-4b89-87f5-ed71964cde2c}
   Method M_Stopping: Id {72700132-7159-42d1-9da3-fac2d393e036}
   Method M_Suspended: Id {073e1932-7551-4d55-960b-702ab8915955}
   Method M_Suspending: Id {41298518-d022-4fd2-814a-dab820629ffd}
   Method M_Undefined: Id {58755443-af9d-4d3e-aca7-a634b5941bbb}
   Method M_Unholding: Id {2d1c0a06-196f-4f18-a8b4-e49409c39881}
   Method M_Unsuspending: Id {0b99b7cd-e845-4aec-8993-abd7fcf7e532}
   Method MandrelCalibration: Id {39c6017d-3381-4a9f-8bc6-c60e36adbd56}
   Property MandrelVacuum: Id {daad43ef-8d3d-4d99-bc52-f75f95baf184}
   Get Get: Id {f61f4ab4-fac0-4178-bdf9-a05c369b6b8c}
   Set Set: Id {97015efa-dd25-4e34-bd76-a318500ce5ef}
   Method ReadParameters: Id {e2e0a2dc-167d-49c5-8f59-82df96707744}
   Method SaveParameters: Id {9b2a545f-584b-4c00-8d82-f9848d7b9196} *)
